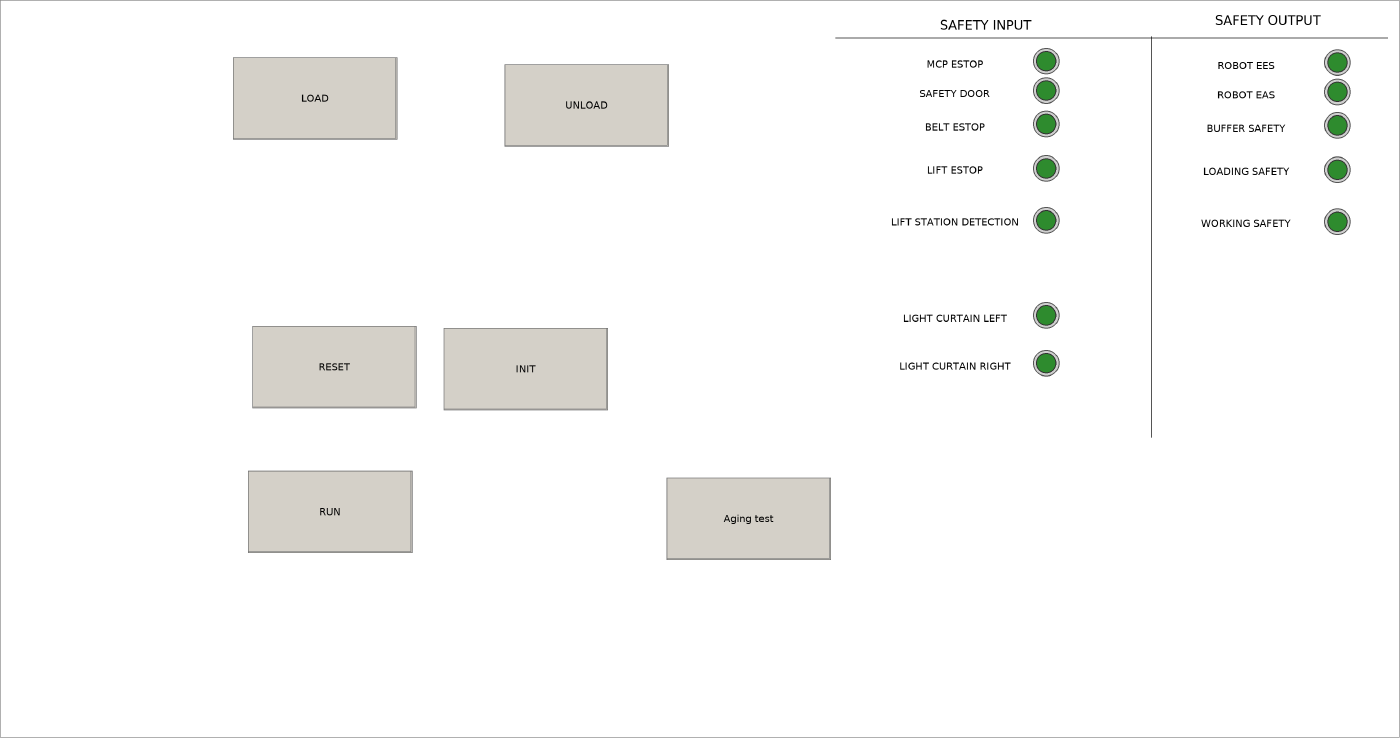
VISUALIZATION visu_operation  // 2048x1080
    Button (369,477 240x120), "RESET", colour toggle: G_HMI.bReset
        OnMouseDown: execute { G_HMI.bReset	:= TRUE; }
        OnMouseUp: execute { G_HMI.bReset	:= FALSE; }
    Button (363,689 240x120), "RUN", colour toggle: G_HMI.bRun
        OnMouseDown: execute { G_HMI.bRun	:= TRUE; }
        OnMouseUp: execute { G_HMI.bRun	:= FALSE; }
    Button (649,480 240x120), "INIT", colour toggle: G_HMI.bInit
        OnMouseDown: execute { G_HMI.bInit	:= TRUE; }
        OnMouseUp: execute { G_HMI.bInit	:= FALSE; }
    Lamp1 (1508,67 45x45), variable: MAIN.application.safety.mcp_estop, style: Lamp-Lamp1-Green
    Label (1287,79 220x30), "MCP ESTOP"
    Lamp1 (1508,159 45x45), variable: MAIN.application.safety.belt_estop, style: Lamp-Lamp1-Green
    Label (1287,171 220x30), "BELT ESTOP"
    Lamp1 (1508,224 45x45), variable: MAIN.application.safety.lift_estop, style: Lamp-Lamp1-Green
    Label (1287,236 220x26), "LIFT ESTOP"
    Lamp1 (1508,300 45x45), variable: MAIN.application.safety.lift_station_detection, style: Lamp-Lamp1-Green
    Label (1287,312 220x26), "LIFT STATION DETECTION"
    Lamp1 (1508,110 45x45), variable: MAIN.application.safety.mcp_safetyDoor, style: Lamp-Lamp1-Green
    Label (1287,122 220x30), "SAFETY DOOR"
    Lamp1 (1508,439 45x45), variable: MAIN.application.safety.lift_lightCurtain_left, style: Lamp-Lamp1-Green
    Label (1287,451 220x30), "LIGHT CURTAIN LEFT"
    Lamp1 (1508,509 45x45), variable: MAIN.application.safety.lift_lightCurtain_right, style: Lamp-Lamp1-Green
    Label (1287,521 220x30), "LIGHT CURTAIN RIGHT"
    Lamp1 (1934,69 45x45), variable: MAIN.application.safety.robot_EES, style: Lamp-Lamp1-Green
    Label (1713,81 220x30), "ROBOT EES"
    Lamp1 (1934,161 45x45), variable: MAIN.application.safety.buffer_safety, style: Lamp-Lamp1-Green
    Label (1713,173 220x30), "BUFFER SAFETY"
    Lamp1 (1934,226 45x45), variable: MAIN.application.safety.loding_safety, style: Lamp-Lamp1-Green
    Label (1713,238 220x26), "LOADING SAFETY"
    Lamp1 (1934,302 45x45), variable: MAIN.application.safety.working_safety, style: Lamp-Lamp1-Green
    Label (1713,314 220x26), "WORKING SAFETY"
    Lamp1 (1934,112 45x45), variable: MAIN.application.safety.robot_EAS, style: Lamp-Lamp1-Green
    Label (1713,124 220x30), "ROBOT EAS"
    Line (1684,640) (1684,53)
    Label (1332,22 220x30), "SAFETY INPUT"
    Label (1745,15 220x30), "SAFETY OUTPUT"
    Line (1222,55) (2030,55)
    Button (341,84 240x120), "LOAD"
        OnMouseDown: execute { MAIN.application.tote_subsystem.cmd	:= OrderToteCommand.LOAD; }
        OnMouseUp: execute {  }
    Button (738,94 240x120), "UNLOAD"
        OnMouseDown: execute { MAIN.application.tote_subsystem.cmd	:= OrderToteCommand.UNLOAD; }
        OnMouseUp: execute {  }
    Button (975,699 240x120), "Aging test", colour toggle: G_HMI.bAging_test
        OnMouseDown: execute { G_HMI.bAging_test	:= TRUE; }
        OnMouseUp: execute { G_HMI.bAging_test	:= FALSE; }
END_VISUALIZATION

(* stored: Version 1.1.0.1, ProductVersion 3.1.4024.12
   Visu visu_operation: Id {4abbf3f6-c173-4bcb-82b6-c0f3163ef68d} *)
